Universal Robots PolyScope program: cinta.2.urp

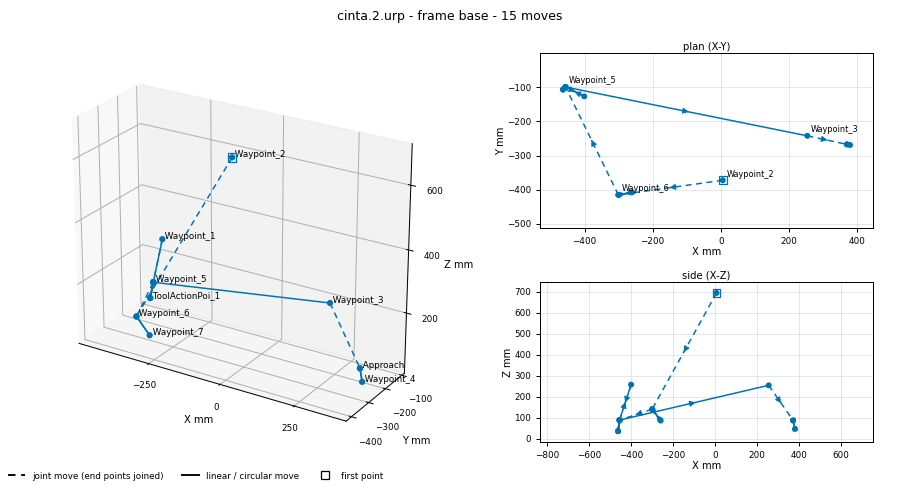
[picture p0: tool path of cinta.2.urp in frame base, 15 of 15 moves have a stored position in this frame; points joined in program order, loops and branches not executed]
Program cinta.2 (installation=default directory=/programs createdIn=5.14.5 lastSavedIn=5.14.5 robotSerialNumber=20195300809)
Calibrated DH parameters: a=[-0.000085, -0.20076, -0.212369, 0.000121, -0.000118, 0]; d=[0.15185, -26.306375, 24.753047, 1.684739, 0.085386, 0.092088]; alpha=[1.572149, -0.00522, -0.011864, 1.571339, -1.571085, 0]; deltaTheta=[0, 0.599885, -0.513355, -0.086555, 0.000006, 0]
InitVariablesNode variables(variable(name=Pallet_1_cnt_1, expression=1), variable(name=Pallet_1_lct, expression=1), variable(name=Pallet_1_lno, expression=1), variable(name=Pallet_1_sep, expression=False), variable(name=Pallet_1_tct, expression=1), variable(name=Pallet_2_cnt_1, expression=1), variable(name=Pallet_2_cnt_2, expression=1), variable(name=Pallet_2_lct, expression=1), variable(name=Pallet_2_lct_1, expression=1), variable(name=Pallet_2_lno, expression=1), variable(name=Pallet_2_lno_1, expression=1), variable(name=Pallet_2_sep, expression=False), variable(name=Pallet_2_sep_1, expression=False), variable(name=Pallet_2_tct, expression=1), variable(name=Pallet_2_tct_1, expression=1), variable(name=Pallet_4_cnt, expression=1), variable(name=Pallet_4_lct, expression=1), variable(name=Pallet_4_lno, expression=1), variable(name=Pallet_4_sep, expression=False), variable(name=Pallet_4_tct, expression=1))
Robot Program (runOnlyOnce=false)
  URCap Gripper Activate (Robotiq_Grippers, Robotiq Inc.) dataModel(ResetAndActivateKey=false)
  MoveJ speed 60 deg/s, acceleration 80 deg/s^2 (useActiveTCP=true) feature=Base
    Waypoint Waypoint_2: TCP in base x=5.936 y=-372.7 z=694.672 mm, rx=-0.0178 ry=2.2101 rz=-2.2165 rad; joints [0.003, -89.998, 0.001, -89.999, 0, 0.002] deg; TCP offset x=0 y=0 z=150 mm, rx=0 ry=0 rz=0 rad
  Wait DigitalInput pin=digital_in[0]; digitalValue=0
  URCap Palletizing (polyscope-pallet-impl, Universal Robots) dataModel(palletFeature=Base, isPalletizing=true, Variable(key=name, variable(name=Pallet_1)), Variable(key=globalCountingVariable, variable(name=Pallet_1_cnt_1, initializeExpression=1)), Variable(key=layerNumberVariable, variable(name=Pallet_1_lno, initializeExpression=1)), Variable(key=layerCountingVariable, variable(name=Pallet_1_lct, initializeExpression=1)), Variable(key=handleSeparatorVariable, variable(name=Pallet_1_sep, initializeExpression=False)), Variable(key=totalCountVariable, variable(name=Pallet_1_tct, initializeExpression=1)), Length(key=objectHeight value=0.04 unit=M), Variable(key=referencePoint, variable(featureName=referencePoint)), Variable(key=separatorPoint, variable(featureName=separatorPoint))); state(isChildrenLocked=true)
    URCap Patterns (polyscope-pallet-impl, Universal Robots) state(isChildrenLocked=true)
      URCap Pattern (polyscope-pallet-impl, Universal Robots) dataModel(UUID=7d18734c-cb0f-4b21-a534-5904a56affce, patternType=IRREGULAR, Variable(key=nameVariable, variable(name=Irreg_Pattern_1))); state(isChildrenLocked=true)
        URCap Item (polyscope-pallet-impl, Universal Robots) dataModel(UUID=f348ba63-6d21-43bb-8ae8-3964627112de, patternType=IRREGULAR, index=0, calibrationDeltaTheta=[2.0871938292282843E-8, 0.5998849625986696, -0.513354759222901, -0.08655474087847535, 6.239817607139875E-6, -6.658617090343766E-8], calibrationA=[-8.52060452638757E-5, -0.2007601879611388, -0.2123691625519033, 1.2105607098011576E-4, -1.1833705743435544E-4, 0.0], calibrationD=[0.15184970286177432, -26.306374840159272, 24.75304670983349, 1.6847390881089916, 0.085385969004481, 0.09208826337351553], calibrationAlpha=[1.5721487795181908, -0.005219907129425837, -0.011864150755780208, 1.5713392161993658, -1.5710853432049288, 0.0], calibrationJointChecksum=[-1860213401, -1859864814, -1494669377, -1328152407, -1329437658, -1329056899], calibrationStatus=2, calibrationValidChecksum=true, baseToFeature=[0.0, 0.0, 0.0, 0.0, 0.0, 0.0], TCPOffset=[9.391397651714595E-6, 1.2583319936476656E-5, 0.15002059384390531, -4.260528976040452E-5, 2.8840070067630035E-6, -1.0843116676403497E-6], Variable(key=variable, variable(name=Item_1)), JointPositions(key=jointpositions, JointPosition(key=[1], Angle(key=pos value=0.595677 unit=RAD)), JointPosition(key=[2], Angle(key=pos value=-0.675595 unit=RAD)), JointPosition(key=[3], Angle(key=pos value=0.603004 unit=RAD)), JointPosition(key=[4], Angle(key=pos value=-1.618024 unit=RAD)), JointPosition(key=[5], Angle(key=pos value=-1.472761 unit=RAD)), JointPosition(key=[6], Angle(key=pos value=-0.97685 unit=RAD))))
    URCap Layers (polyscope-pallet-impl, Universal Robots) dataModel(separators=[false], selectedPatterns=[7d18734c-cb0f-4b21-a534-5904a56affce])
    URCap At Each Item (polyscope-pallet-impl, Universal Robots) dataModel(selectedPattern=7d18734c-cb0f-4b21-a534-5904a56affce, selectedPosition=f348ba63-6d21-43bb-8ae8-3964627112de, Approach_calibrationDeltaTheta=[2.0871938292282843E-8, 0.5998849625986696, -0.513354759222901, -0.08655474087847535, 6.239817607139875E-6, -6.658617090343766E-8], Approach_calibrationA=[-8.52060452638757E-5, -0.2007601879611388, -0.2123691625519033, 1.2105607098011576E-4, -1.1833705743435544E-4, 0.0], Approach_calibrationD=[0.15184970286177432, -26.306374840159272, 24.75304670983349, 1.6847390881089916, 0.085385969004481, 0.09208826337351553], Approach_calibrationAlpha=[1.5721487795181908, -0.005219907129425837, -0.011864150755780208, 1.5713392161993658, -1.5710853432049288, 0.0], Approach_calibrationJointChecksum=[-1860213401, -1859864814, -1494669377, -1328152407, -1329437658, -1329056899], Approach_calibrationStatus=2, Approach_calibrationValidChecksum=true, Approach_baseToFeature=[0.0, 0.0, 0.0, 0.0, 0.0, 0.0], Approach_TCPOffset=[6.288453330560717E-6, -4.440500703251082E-6, 0.14999119071126726, 5.857466069426218E-5, -5.428145810996883E-6, 2.090200739322049E-5], Exit_calibrationDeltaTheta=[2.0871938292282843E-8, 0.5998849625986696, -0.513354759222901, -0.08655474087847535, 6.239817607139875E-6, -6.658617090343766E-8], Exit_calibrationA=[-8.52060452638757E-5, -0.2007601879611388, -0.2123691625519033, 1.2105607098011576E-4, -1.1833705743435544E-4, 0.0], Exit_calibrationD=[0.15184970286177432, -26.306374840159272, 24.75304670983349, 1.6847390881089916, 0.085385969004481, 0.09208826337351553], Exit_calibrationAlpha=[1.5721487795181908, -0.005219907129425837, -0.011864150755780208, 1.5713392161993658, -1.5710853432049288, 0.0], Exit_calibrationJointChecksum=[-1860213401, -1859864814, -1494669377, -1328152407, -1329437658, -1329056899], Exit_calibrationStatus=2, Exit_calibrationValidChecksum=true, Exit_baseToFeature=[0.0, 0.0, 0.0, 0.0, 0.0, 0.0], Exit_TCPOffset=[-1.7989367446957782E-5, -1.0560005302862052E-5, 0.15002098103245548, -3.476895864800672E-6, -4.621995147941492E-5, -3.533771160372287E-5], currentWizardState=LANDING, Pose(key=refBaseToFeature, Position(key=posePosition, Length(key=X value=0 unit=M), Length(key=Y value=0 unit=M), Length(key=Z value=0 unit=M)), Rotation(key=poseRotation, Angle(key=RX value=0 unit=RAD), Angle(key=RY value=0 unit=RAD), Angle(key=RZ value=0 unit=RAD))), Pose(key=refPose, Position(key=posePosition, Length(key=X value=-0.356569 unit=M), Length(key=Y value=-0.423777 unit=M), Length(key=Z value=0.09165 unit=M)), Rotation(key=poseRotation, Angle(key=RX value=0.142297 unit=RAD), Angle(key=RY value=-3.021243 unit=RAD), Angle(key=RZ value=0.176168 unit=RAD))), JointPositions(key=Approach_jointpositions, JointPosition(key=[1], Angle(key=pos value=0.546001 unit=RAD)), JointPosition(key=[2], Angle(key=pos value=-0.682183 unit=RAD)), JointPosition(key=[3], Angle(key=pos value=0.323504 unit=RAD)), JointPosition(key=[4], Angle(key=pos value=-1.411958 unit=RAD)), JointPosition(key=[5], Angle(key=pos value=-1.400218 unit=RAD)), JointPosition(key=[6], Angle(key=pos value=-1.026097 unit=RAD))), JointPositions(key=Exit_jointpositions, JointPosition(key=[1], Angle(key=pos value=0.615816 unit=RAD)), JointPosition(key=[2], Angle(key=pos value=-0.58775 unit=RAD)), JointPosition(key=[3], Angle(key=pos value=0.453411 unit=RAD)), JointPosition(key=[4], Angle(key=pos value=-1.593643 unit=RAD)), JointPosition(key=[5], Angle(key=pos value=-1.548909 unit=RAD)), JointPosition(key=[6], Angle(key=pos value=-1.048656 unit=RAD))))
      URCap Generated Movements (polyscope-pallet-impl, Universal Robots) state(isChildrenLocked=true)
        MoveJ speed 60 deg/s, acceleration 80 deg/s^2 (useActiveTCP=true) feature=referencePoint
          Waypoint Waypoint_6: TCP in base x=-300.88 y=-415.654 z=140.629 mm, rx=-0.0198 ry=-3.0249 rz=0.2808 rad; joints [36.906, -52.821, 49.281, -97.642, -86.084, -51.998] deg; feature pose in base x=-356.569 y=-423.777 z=91.65 mm, rx=0.1423 ry=-3.0212 rz=0.1762 rad
        MoveL speed 250 mm/s, acceleration 1200 mm/s^2 (useActiveTCP=true) feature(featureName=referencePoint)
          Waypoint Waypoint_7: TCP in base x=-260.278 y=-408.079 z=86.393 mm, rx=-0.0542 ry=-3.111 rz=0.0452 rad; joints [41.67, -49.638, 53.512, -96.276, -90.815, -46.427] deg
          SetPayload (workpieceName=Payload)
        Folder Tool action
          URCap Gripper (Robotiq_Grippers, Robotiq Inc.) dataModel(position=100.0, force=5.0, speed=100.0, positionInDouble=100.0, forceInDouble=5.0, speedInDouble=100.0, slaveIds=[3], blocking=true)
        MoveL speed 250 mm/s, acceleration 1200 mm/s^2 (useActiveTCP=true) feature(featureName=referencePoint)
          Waypoint Waypoint_6: TCP in base x=-300.88 y=-415.654 z=140.629 mm, rx=-0.0198 ry=-3.0249 rz=0.2808 rad; joints [36.906, -52.821, 49.281, -97.642, -86.084, -51.998] deg
  URCap Palletizing (polyscope-pallet-impl, Universal Robots) dataModel(palletFeature=Base, isPalletizing=false, Variable(key=name, variable(name=Pallet_2)), Variable(key=globalCountingVariable, variable(name=Pallet_2_cnt_1, initializeExpression=1)), Variable(key=layerNumberVariable, variable(name=Pallet_2_lno, initializeExpression=1)), Variable(key=layerCountingVariable, variable(name=Pallet_2_lct, initializeExpression=1)), Variable(key=handleSeparatorVariable, variable(name=Pallet_2_sep, initializeExpression=False)), Variable(key=totalCountVariable, variable(name=Pallet_2_tct, initializeExpression=1)), Length(key=objectHeight value=0.05 unit=M), Variable(key=referencePoint, variable(featureName=referencePoin_1)), Variable(key=separatorPoint, variable(featureName=separatorPoin_1))); state(isChildrenLocked=true)
    URCap Patterns (polyscope-pallet-impl, Universal Robots) state(isChildrenLocked=true)
      URCap Pattern (polyscope-pallet-impl, Universal Robots) dataModel(UUID=70c9da9f-f26c-40af-87f5-4ef85564398c, patternType=IRREGULAR, Variable(key=nameVariable, variable(name=Irreg_Pattern_2))); state(isChildrenLocked=true)
        URCap Item (polyscope-pallet-impl, Universal Robots) dataModel(UUID=c27a4a84-36a7-4a3e-9bbe-b9e4806bb6c1, patternType=IRREGULAR, index=0, calibrationDeltaTheta=[2.0871938292282843E-8, 0.5998849625986696, -0.513354759222901, -0.08655474087847535, 6.239817607139875E-6, -6.658617090343766E-8], calibrationA=[-8.52060452638757E-5, -0.2007601879611388, -0.2123691625519033, 1.2105607098011576E-4, -1.1833705743435544E-4, 0.0], calibrationD=[0.15184970286177432, -26.306374840159272, 24.75304670983349, 1.6847390881089916, 0.085385969004481, 0.09208826337351553], calibrationAlpha=[1.5721487795181908, -0.005219907129425837, -0.011864150755780208, 1.5713392161993658, -1.5710853432049288, 0.0], calibrationJointChecksum=[-1860213401, -1859864814, -1494669377, -1328152407, -1329437658, -1329056899], calibrationStatus=2, calibrationValidChecksum=true, baseToFeature=[0.0, 0.0, 0.0, 0.0, 0.0, 0.0], TCPOffset=[1.4796052247856295E-6, -1.2520157244955143E-5, 0.14999059913150856, 4.686731117752855E-5, -3.293405451311865E-5, 2.7796227253080194E-5], Variable(key=variable, variable(name=Item_2)), JointPositions(key=jointpositions, JointPosition(key=[1], Angle(key=pos value=-0.101307 unit=RAD)), JointPosition(key=[2], Angle(key=pos value=-0.846515 unit=RAD)), JointPosition(key=[3], Angle(key=pos value=1.123983 unit=RAD)), JointPosition(key=[4], Angle(key=pos value=-1.842057 unit=RAD)), JointPosition(key=[5], Angle(key=pos value=-1.498402 unit=RAD)), JointPosition(key=[6], Angle(key=pos value=-0.155893 unit=RAD))))
    URCap Layers (polyscope-pallet-impl, Universal Robots) dataModel(separators=[false], selectedPatterns=[70c9da9f-f26c-40af-87f5-4ef85564398c])
    URCap At Each Item (polyscope-pallet-impl, Universal Robots) dataModel(selectedPattern=70c9da9f-f26c-40af-87f5-4ef85564398c, selectedPosition=c27a4a84-36a7-4a3e-9bbe-b9e4806bb6c1, Approach_calibrationDeltaTheta=[2.0871938292282843E-8, 0.5998849625986696, -0.513354759222901, -0.08655474087847535, 6.239817607139875E-6, -6.658617090343766E-8], Approach_calibrationA=[-8.52060452638757E-5, -0.2007601879611388, -0.2123691625519033, 1.2105607098011576E-4, -1.1833705743435544E-4, 0.0], Approach_calibrationD=[0.15184970286177432, -26.306374840159272, 24.75304670983349, 1.6847390881089916, 0.085385969004481, 0.09208826337351553], Approach_calibrationAlpha=[1.5721487795181908, -0.005219907129425837, -0.011864150755780208, 1.5713392161993658, -1.5710853432049288, 0.0], Approach_calibrationJointChecksum=[-1860213401, -1859864814, -1494669377, -1328152407, -1329437658, -1329056899], Approach_calibrationStatus=2, Approach_calibrationValidChecksum=true, Approach_baseToFeature=[0.0, 0.0, 0.0, 0.0, 0.0, 0.0], Approach_TCPOffset=[-2.435285091917372E-6, -2.2477675725607327E-5, 0.14996372139900316, 1.2485897723616868E-4, 1.936593107412943E-5, -3.0361418856762723E-5], Exit_calibrationDeltaTheta=[2.0871938292282843E-8, 0.5998849625986696, -0.513354759222901, -0.08655474087847535, 6.239817607139875E-6, -6.658617090343766E-8], Exit_calibrationA=[-8.52060452638757E-5, -0.2007601879611388, -0.2123691625519033, 1.2105607098011576E-4, -1.1833705743435544E-4, 0.0], Exit_calibrationD=[0.15184970286177432, -26.306374840159272, 24.75304670983349, 1.6847390881089916, 0.085385969004481, 0.09208826337351553], Exit_calibrationAlpha=[1.5721487795181908, -0.005219907129425837, -0.011864150755780208, 1.5713392161993658, -1.5710853432049288, 0.0], Exit_calibrationJointChecksum=[-1860213401, -1859864814, -1494669377, -1328152407, -1329437658, -1329056899], Exit_calibrationStatus=2, Exit_calibrationValidChecksum=true, Exit_baseToFeature=[0.0, 0.0, 0.0, 0.0, 0.0, 0.0], Exit_TCPOffset=[1.7062831376105092E-5, 3.524481410888125E-6, 0.1500131622037378, -3.3427689265285523E-5, -7.770367597523134E-6, 3.124336029970859E-5], currentWizardState=LANDING, Pose(key=refBaseToFeature, Position(key=posePosition, Length(key=X value=0 unit=M), Length(key=Y value=0 unit=M), Length(key=Z value=0 unit=M)), Rotation(key=poseRotation, Angle(key=RX value=0 unit=RAD), Angle(key=RY value=0 unit=RAD), Angle(key=RZ value=0 unit=RAD))), Pose(key=refPose, Position(key=posePosition, Length(key=X value=-0.463666 unit=M), Length(key=Y value=-0.106221 unit=M), Length(key=Z value=0.035787 unit=M)), Rotation(key=poseRotation, Angle(key=RX value=2.122927 unit=RAD), Angle(key=RY value=2.233822 unit=RAD), Angle(key=RZ value=-0.100576 unit=RAD))), JointPositions(key=Approach_jointpositions, JointPosition(key=[1], Angle(key=pos value=-0.083249 unit=RAD)), JointPosition(key=[2], Angle(key=pos value=-0.988428 unit=RAD)), JointPosition(key=[3], Angle(key=pos value=1.052561 unit=RAD)), JointPosition(key=[4], Angle(key=pos value=-1.655373 unit=RAD)), JointPosition(key=[5], Angle(key=pos value=-1.48077 unit=RAD)), JointPosition(key=[6], Angle(key=pos value=-0.155884 unit=RAD))), JointPositions(key=Exit_jointpositions, JointPosition(key=[1], Angle(key=pos value=-0.101329 unit=RAD)), JointPosition(key=[2], Angle(key=pos value=-0.846523 unit=RAD)), JointPosition(key=[3], Angle(key=pos value=1.123971 unit=RAD)), JointPosition(key=[4], Angle(key=pos value=-1.842077 unit=RAD)), JointPosition(key=[5], Angle(key=pos value=-1.498362 unit=RAD)), JointPosition(key=[6], Angle(key=pos value=-0.155884 unit=RAD))))
      URCap Generated Movements (polyscope-pallet-impl, Universal Robots) state(isChildrenLocked=true)
        MoveJ speed 60 deg/s, acceleration 80 deg/s^2 (useActiveTCP=true) feature=referencePoin_1
          Waypoint Waypoint_5: TCP in base x=-456.282 y=-98.651 z=88.709 mm, rx=2.1005 ry=2.2182 rz=-0.0592 rad; joints [-6.749, -50.646, 52.859, -89.594, -86.16, -9.971] deg; feature pose in base x=-463.666 y=-106.221 z=35.787 mm, rx=2.1229 ry=2.2338 rz=-0.1006 rad
        MoveL speed 250 mm/s, acceleration 1200 mm/s^2 (useActiveTCP=true) feature(featureName=referencePoin_1)
          Waypoint ToolActionPoi_1: TCP in base x=-463.666 y=-106.221 z=35.787 mm, rx=2.1229 ry=2.2338 rz=-0.1006 rad; joints [-5.804, -48.502, 64.399, -105.542, -85.852, -8.932] deg; TCP offset x=0.001 y=-0.013 z=149.991 mm, rx=0 ry=0 rz=0 rad
        Folder Tool action
          URCap Gripper (Robotiq_Grippers, Robotiq Inc.) dataModel(position=0.0, force=100.0, speed=100.0, positionInDouble=0.0, forceInDouble=100.0, speedInDouble=100.0, slaveIds=[3], blocking=true)
        MoveL speed 250 mm/s, acceleration 1200 mm/s^2 (useActiveTCP=true) feature(featureName=referencePoin_1)
          Waypoint Waypoint_5: TCP in base x=-456.282 y=-98.651 z=88.709 mm, rx=2.1005 ry=2.2182 rz=-0.0592 rad; joints [-6.749, -50.646, 52.859, -89.594, -86.16, -9.971] deg; TCP offset x=0 y=0 z=150 mm, rx=0 ry=0 rz=0 rad
  MoveL speed 250 mm/s, acceleration 1200 mm/s^2 (useActiveTCP=true) feature=Base
    Waypoint Waypoint_1: TCP in base x=-401.164 y=-126.147 z=257.714 mm, rx=-2.0401 ry=-2.1933 rz=0.3328 rad; joints [-4.037, -76.934, 54.545, -81.338, -85.663, -7.38] deg
  Wait Sleep waitTime=3
  URCap Palletizing (polyscope-pallet-impl, Universal Robots) dataModel(palletFeature=Base, isPalletizing=false, Length(key=objectHeight value=0.05 unit=M), Variable(key=name, variable(name=Pallet_3)), Variable(key=globalCountingVariable, variable(name=Pallet_2_cnt_2, initializeExpression=1)), Variable(key=layerCountingVariable, variable(name=Pallet_2_lct_1, initializeExpression=1)), Variable(key=layerNumberVariable, variable(name=Pallet_2_lno_1, initializeExpression=1)), Variable(key=handleSeparatorVariable, variable(name=Pallet_2_sep_1, initializeExpression=False)), Variable(key=totalCountVariable, variable(name=Pallet_2_tct_1, initializeExpression=1)), Variable(key=referencePoint, variable(featureName=referencePoin_2)), Variable(key=separatorPoint, variable(featureName=separatorPoin_2))); state(isChildrenLocked=true)
    URCap Patterns (polyscope-pallet-impl, Universal Robots) state(isChildrenLocked=true)
      URCap Pattern (polyscope-pallet-impl, Universal Robots) dataModel(UUID=70c9da9f-f26c-40af-87f5-4ef85564398c, patternType=IRREGULAR, Variable(key=nameVariable, variable(name=Irreg_Pattern_3))); state(isChildrenLocked=true)
        URCap Item (polyscope-pallet-impl, Universal Robots) dataModel(UUID=c27a4a84-36a7-4a3e-9bbe-b9e4806bb6c1, patternType=IRREGULAR, index=0, calibrationDeltaTheta=[2.0871938292282843E-8, 0.5998849625986696, -0.513354759222901, -0.08655474087847535, 6.239817607139875E-6, -6.658617090343766E-8], calibrationA=[-8.52060452638757E-5, -0.2007601879611388, -0.2123691625519033, 1.2105607098011576E-4, -1.1833705743435544E-4, 0.0], calibrationD=[0.15184970286177432, -26.306374840159272, 24.75304670983349, 1.6847390881089916, 0.085385969004481, 0.09208826337351553], calibrationAlpha=[1.5721487795181908, -0.005219907129425837, -0.011864150755780208, 1.5713392161993658, -1.5710853432049288, 0.0], calibrationJointChecksum=[-1860213401, -1859864814, -1494669377, -1328152407, -1329437658, -1329056899], calibrationStatus=2, calibrationValidChecksum=true, baseToFeature=[0.0, 0.0, 0.0, 0.0, 0.0, 0.0], TCPOffset=[1.4796052247856295E-6, -1.2520157244955143E-5, 0.14999059913150856, 4.686731117752855E-5, -3.293405451311865E-5, 2.7796227253080194E-5], JointPositions(key=jointpositions, JointPosition(key=[1], Angle(key=pos value=-0.101307 unit=RAD)), JointPosition(key=[2], Angle(key=pos value=-0.846515 unit=RAD)), JointPosition(key=[3], Angle(key=pos value=1.123983 unit=RAD)), JointPosition(key=[4], Angle(key=pos value=-1.842057 unit=RAD)), JointPosition(key=[5], Angle(key=pos value=-1.498402 unit=RAD)), JointPosition(key=[6], Angle(key=pos value=-0.155893 unit=RAD))), Variable(key=variable, variable(name=Item_3)))
    URCap Layers (polyscope-pallet-impl, Universal Robots) dataModel(separators=[false], selectedPatterns=[70c9da9f-f26c-40af-87f5-4ef85564398c])
    URCap At Each Item (polyscope-pallet-impl, Universal Robots) dataModel(selectedPattern=70c9da9f-f26c-40af-87f5-4ef85564398c, selectedPosition=c27a4a84-36a7-4a3e-9bbe-b9e4806bb6c1, Approach_calibrationDeltaTheta=[2.0871938292282843E-8, 0.5998849625986696, -0.513354759222901, -0.08655474087847535, 6.239817607139875E-6, -6.658617090343766E-8], Approach_calibrationA=[-8.52060452638757E-5, -0.2007601879611388, -0.2123691625519033, 1.2105607098011576E-4, -1.1833705743435544E-4, 0.0], Approach_calibrationD=[0.15184970286177432, -26.306374840159272, 24.75304670983349, 1.6847390881089916, 0.085385969004481, 0.09208826337351553], Approach_calibrationAlpha=[1.5721487795181908, -0.005219907129425837, -0.011864150755780208, 1.5713392161993658, -1.5710853432049288, 0.0], Approach_calibrationJointChecksum=[-1860213401, -1859864814, -1494669377, -1328152407, -1329437658, -1329056899], Approach_calibrationStatus=2, Approach_calibrationValidChecksum=true, Approach_baseToFeature=[0.0, 0.0, 0.0, 0.0, 0.0, 0.0], Approach_TCPOffset=[-2.435285091917372E-6, -2.2477675725607327E-5, 0.14996372139900316, 1.2485897723616868E-4, 1.936593107412943E-5, -3.0361418856762723E-5], Exit_calibrationDeltaTheta=[2.0871938292282843E-8, 0.5998849625986696, -0.513354759222901, -0.08655474087847535, 6.239817607139875E-6, -6.658617090343766E-8], Exit_calibrationA=[-8.52060452638757E-5, -0.2007601879611388, -0.2123691625519033, 1.2105607098011576E-4, -1.1833705743435544E-4, 0.0], Exit_calibrationD=[0.15184970286177432, -26.306374840159272, 24.75304670983349, 1.6847390881089916, 0.085385969004481, 0.09208826337351553], Exit_calibrationAlpha=[1.5721487795181908, -0.005219907129425837, -0.011864150755780208, 1.5713392161993658, -1.5710853432049288, 0.0], Exit_calibrationJointChecksum=[-1860213401, -1859864814, -1494669377, -1328152407, -1329437658, -1329056899], Exit_calibrationStatus=2, Exit_calibrationValidChecksum=true, Exit_baseToFeature=[0.0, 0.0, 0.0, 0.0, 0.0, 0.0], Exit_TCPOffset=[1.7062831376105092E-5, 3.524481410888125E-6, 0.1500131622037378, -3.3427689265285523E-5, -7.770367597523134E-6, 3.124336029970859E-5], currentWizardState=LANDING, Pose(key=refBaseToFeature, Position(key=posePosition, Length(key=X value=0 unit=M), Length(key=Y value=0 unit=M), Length(key=Z value=0 unit=M)), Rotation(key=poseRotation, Angle(key=RX value=0 unit=RAD), Angle(key=RY value=0 unit=RAD), Angle(key=RZ value=0 unit=RAD))), Pose(key=refPose, Position(key=posePosition, Length(key=X value=-0.463666 unit=M), Length(key=Y value=-0.106221 unit=M), Length(key=Z value=0.035787 unit=M)), Rotation(key=poseRotation, Angle(key=RX value=2.122927 unit=RAD), Angle(key=RY value=2.233822 unit=RAD), Angle(key=RZ value=-0.100576 unit=RAD))), JointPositions(key=Approach_jointpositions, JointPosition(key=[1], Angle(key=pos value=-0.083249 unit=RAD)), JointPosition(key=[2], Angle(key=pos value=-0.988428 unit=RAD)), JointPosition(key=[3], Angle(key=pos value=1.052561 unit=RAD)), JointPosition(key=[4], Angle(key=pos value=-1.655373 unit=RAD)), JointPosition(key=[5], Angle(key=pos value=-1.48077 unit=RAD)), JointPosition(key=[6], Angle(key=pos value=-0.155884 unit=RAD))), JointPositions(key=Exit_jointpositions, JointPosition(key=[1], Angle(key=pos value=-0.101329 unit=RAD)), JointPosition(key=[2], Angle(key=pos value=-0.846523 unit=RAD)), JointPosition(key=[3], Angle(key=pos value=1.123971 unit=RAD)), JointPosition(key=[4], Angle(key=pos value=-1.842077 unit=RAD)), JointPosition(key=[5], Angle(key=pos value=-1.498362 unit=RAD)), JointPosition(key=[6], Angle(key=pos value=-0.155884 unit=RAD))))
      URCap Generated Movements (polyscope-pallet-impl, Universal Robots) state(isChildrenLocked=true)
        MoveJ speed 60 deg/s, acceleration 80 deg/s^2 (useActiveTCP=true) feature=referencePoin_2
          Waypoint Waypoint_5: TCP in base x=-456.282 y=-98.651 z=88.709 mm, rx=2.1005 ry=2.2182 rz=-0.0592 rad; joints [-6.749, -50.646, 52.859, -89.594, -86.16, -9.971] deg; feature pose in base x=-463.666 y=-106.221 z=35.787 mm, rx=2.1229 ry=2.2338 rz=-0.1006 rad
        MoveL speed 250 mm/s, acceleration 1200 mm/s^2 (useActiveTCP=true) feature(featureName=referencePoin_2)
          Waypoint ToolActionPoi_1: TCP in base x=-463.666 y=-106.221 z=35.787 mm, rx=2.1229 ry=2.2338 rz=-0.1006 rad; joints [-5.804, -48.502, 64.399, -105.542, -85.852, -8.932] deg; TCP offset x=0.001 y=-0.013 z=149.991 mm, rx=0 ry=0 rz=0 rad
        Folder Tool action
          URCap Gripper (Robotiq_Grippers, Robotiq Inc.) dataModel(position=100.0, force=5.0, speed=100.0, positionInDouble=100.0, forceInDouble=5.0, speedInDouble=100.0, slaveIds=[3], blocking=true)
        MoveL speed 250 mm/s, acceleration 1200 mm/s^2 (useActiveTCP=true) feature(featureName=referencePoin_2)
          Waypoint Waypoint_5: TCP in base x=-456.282 y=-98.651 z=88.709 mm, rx=2.1005 ry=2.2182 rz=-0.0592 rad; joints [-6.749, -50.646, 52.859, -89.594, -86.16, -9.971] deg; TCP offset x=0 y=0 z=150 mm, rx=0 ry=0 rz=0 rad
  MoveL speed 250 mm/s, acceleration 1200 mm/s^2 (useActiveTCP=true) feature=Base
    Waypoint Waypoint_3: TCP in base x=254.459 y=-242.142 z=254.509 mm, rx=0.8314 ry=-2.8675 rz=0.0376 rad; joints [120.819, -72.018, 40.908, -57.961, -99.758, -0.985] deg
  URCap Palletizing (polyscope-pallet-impl, Universal Robots) dataModel(palletFeature=Base, isPalletizing=true, Variable(key=name, variable(name=Pallet_4)), Variable(key=globalCountingVariable, variable(name=Pallet_4_cnt, initializeExpression=1)), Variable(key=layerNumberVariable, variable(name=Pallet_4_lno, initializeExpression=1)), Variable(key=layerCountingVariable, variable(name=Pallet_4_lct, initializeExpression=1)), Variable(key=handleSeparatorVariable, variable(name=Pallet_4_sep, initializeExpression=False)), Variable(key=totalCountVariable, variable(name=Pallet_4_tct, initializeExpression=1)), Length(key=objectHeight value=0.05 unit=M), Variable(key=referencePoint, variable(featureName=referencePoin_3)), Variable(key=separatorPoint, variable(featureName=separatorPoin_3))); state(isChildrenLocked=true)
    URCap Patterns (polyscope-pallet-impl, Universal Robots) state(isChildrenLocked=true)
      URCap Pattern (polyscope-pallet-impl, Universal Robots) dataModel(UUID=acebaf78-3d78-4eb2-9b5d-84c80f213af3, patternType=GRID, columns=3, rows=2, Variable(key=nameVariable, variable(name=Grid_Pattern_1))); state(isChildrenLocked=true)
        URCap Item (polyscope-pallet-impl, Universal Robots) dataModel(UUID=c01159d7-bdc8-4ad0-a768-e1fc64c23f72, patternType=GRID, index=0, calibrationDeltaTheta=[2.0871938292282843E-8, 0.5998849625986696, -0.513354759222901, -0.08655474087847535, 6.239817607139875E-6, -6.658617090343766E-8], calibrationA=[-8.52060452638757E-5, -0.2007601879611388, -0.2123691625519033, 1.2105607098011576E-4, -1.1833705743435544E-4, 0.0], calibrationD=[0.15184970286177432, -26.306374840159272, 24.75304670983349, 1.6847390881089916, 0.085385969004481, 0.09208826337351553], calibrationAlpha=[1.5721487795181908, -0.005219907129425837, -0.011864150755780208, 1.5713392161993658, -1.5710853432049288, 0.0], calibrationJointChecksum=[-1860213401, -1859864814, -1494669377, -1328152407, -1329437658, -1329056899], calibrationStatus=2, calibrationValidChecksum=true, baseToFeature=[0.0, 0.0, 0.0, 0.0, 0.0, 0.0], TCPOffset=[3.62221013627817E-7, 2.3695177266913614E-5, 0.14997395472124347, -8.099408147510325E-5, 4.151938501836787E-5, 1.2179441318642959E-5], Variable(key=variable, variable(name=CornerItem_1)), JointPositions(key=jointpositions, JointPosition(key=[1], Angle(key=pos value=2.248677 unit=RAD)), JointPosition(key=[2], Angle(key=pos value=-0.912649 unit=RAD)), JointPosition(key=[3], Angle(key=pos value=1.254868 unit=RAD)), JointPosition(key=[4], Angle(key=pos value=-1.946088 unit=RAD)), JointPosition(key=[5], Angle(key=pos value=-1.5722 unit=RAD)), JointPosition(key=[6], Angle(key=pos value=-2.450668 unit=RAD))))
        URCap Item (polyscope-pallet-impl, Universal Robots) dataModel(UUID=2189a120-c5c3-4d1a-9dea-873932fe821a, patternType=GRID, index=1, calibrationDeltaTheta=[2.0871938292282843E-8, 0.5998849625986696, -0.513354759222901, -0.08655474087847535, 6.239817607139875E-6, -6.658617090343766E-8], calibrationA=[-8.52060452638757E-5, -0.2007601879611388, -0.2123691625519033, 1.2105607098011576E-4, -1.1833705743435544E-4, 0.0], calibrationD=[0.15184970286177432, -26.306374840159272, 24.75304670983349, 1.6847390881089916, 0.085385969004481, 0.09208826337351553], calibrationAlpha=[1.5721487795181908, -0.005219907129425837, -0.011864150755780208, 1.5713392161993658, -1.5710853432049288, 0.0], calibrationJointChecksum=[-1860213401, -1859864814, -1494669377, -1328152407, -1329437658, -1329056899], calibrationStatus=2, calibrationValidChecksum=true, baseToFeature=[0.0, 0.0, 0.0, 0.0, 0.0, 0.0], TCPOffset=[6.919455813991782E-6, -1.59324717010495E-5, 0.15001367778842753, 2.9868797252186343E-5, -4.517849279249192E-6, -4.000161446948098E-5], Variable(key=variable, variable(name=CornerItem_2)), JointPositions(key=jointpositions, JointPosition(key=[1], Angle(key=pos value=2.614511 unit=RAD)), JointPosition(key=[2], Angle(key=pos value=-1.15318 unit=RAD)), JointPosition(key=[3], Angle(key=pos value=1.678785 unit=RAD)), JointPosition(key=[4], Angle(key=pos value=-2.080078 unit=RAD)), JointPosition(key=[5], Angle(key=pos value=-1.587274 unit=RAD)), JointPosition(key=[6], Angle(key=pos value=-2.091675 unit=RAD))))
        URCap Item (polyscope-pallet-impl, Universal Robots) dataModel(UUID=21607d58-3b12-46c5-8d2a-9916ff338648, patternType=GRID, index=2, calibrationDeltaTheta=[2.0871938292282843E-8, 0.5998849625986696, -0.513354759222901, -0.08655474087847535, 6.239817607139875E-6, -6.658617090343766E-8], calibrationA=[-8.52060452638757E-5, -0.2007601879611388, -0.2123691625519033, 1.2105607098011576E-4, -1.1833705743435544E-4, 0.0], calibrationD=[0.15184970286177432, -26.306374840159272, 24.75304670983349, 1.6847390881089916, 0.085385969004481, 0.09208826337351553], calibrationAlpha=[1.5721487795181908, -0.005219907129425837, -0.011864150755780208, 1.5713392161993658, -1.5710853432049288, 0.0], calibrationJointChecksum=[-1860213401, -1859864814, -1494669377, -1328152407, -1329437658, -1329056899], calibrationStatus=2, calibrationValidChecksum=true, baseToFeature=[0.0, 0.0, 0.0, 0.0, 0.0, 0.0], TCPOffset=[-4.63084492346999E-6, -4.863462618229231E-6, 0.1499865178152125, -7.754704754451109E-6, 1.2068952613309615E-6, 1.5530771283901447E-5], Variable(key=variable, variable(name=CornerItem_3)), JointPositions(key=jointpositions, JointPosition(key=[1], Angle(key=pos value=2.74226 unit=RAD)), JointPosition(key=[2], Angle(key=pos value=-0.741952 unit=RAD)), JointPosition(key=[3], Angle(key=pos value=0.93023 unit=RAD)), JointPosition(key=[4], Angle(key=pos value=-1.780847 unit=RAD)), JointPosition(key=[5], Angle(key=pos value=-1.58849 unit=RAD)), JointPosition(key=[6], Angle(key=pos value=-1.919331 unit=RAD))))
        URCap Item (polyscope-pallet-impl, Universal Robots) dataModel(UUID=203bc53d-136e-47a2-98ac-824ae0b9f02c, patternType=GRID, index=3, calibrationDeltaTheta=[2.0871938292282843E-8, 0.5998849625986696, -0.513354759222901, -0.08655474087847535, 6.239817607139875E-6, -6.658617090343766E-8], calibrationA=[-8.52060452638757E-5, -0.2007601879611388, -0.2123691625519033, 1.2105607098011576E-4, -1.1833705743435544E-4, 0.0], calibrationD=[0.15184970286177432, -26.306374840159272, 24.75304670983349, 1.6847390881089916, 0.085385969004481, 0.09208826337351553], calibrationAlpha=[1.5721487795181908, -0.005219907129425837, -0.011864150755780208, 1.5713392161993658, -1.5710853432049288, 0.0], calibrationJointChecksum=[-1860213401, -1859864814, -1494669377, -1328152407, -1329437658, -1329056899], calibrationStatus=2, calibrationValidChecksum=true, baseToFeature=[0.0, 0.0, 0.0, 0.0, 0.0, 0.0], TCPOffset=[2.9663871770058137E-6, -2.7200211151962028E-5, 0.15001295968752965, 2.8669519702431683E-5, -3.4484229554148914E-5, -1.2084844145554098E-5], Variable(key=variable, variable(name=CornerItem_4)), JointPositions(key=jointpositions, JointPosition(key=[1], Angle(key=pos value=2.423566 unit=RAD)), JointPosition(key=[2], Angle(key=pos value=-0.509839 unit=RAD)), JointPosition(key=[3], Angle(key=pos value=0.540103 unit=RAD)), JointPosition(key=[4], Angle(key=pos value=-1.69904 unit=RAD)), JointPosition(key=[5], Angle(key=pos value=-1.581203 unit=RAD)), JointPosition(key=[6], Angle(key=pos value=-2.232232 unit=RAD))))
    URCap Layers (polyscope-pallet-impl, Universal Robots) dataModel(separators=[false], selectedPatterns=[acebaf78-3d78-4eb2-9b5d-84c80f213af3])
    URCap At Each Item (polyscope-pallet-impl, Universal Robots) dataModel(selectedPattern=acebaf78-3d78-4eb2-9b5d-84c80f213af3, selectedPosition=c01159d7-bdc8-4ad0-a768-e1fc64c23f72, Approach_calibrationDeltaTheta=[2.0871938292282843E-8, 0.5998849625986696, -0.513354759222901, -0.08655474087847535, 6.239817607139875E-6, -6.658617090343766E-8], Approach_calibrationA=[-8.52060452638757E-5, -0.2007601879611388, -0.2123691625519033, 1.2105607098011576E-4, -1.1833705743435544E-4, 0.0], Approach_calibrationD=[0.15184970286177432, -26.306374840159272, 24.75304670983349, 1.6847390881089916, 0.085385969004481, 0.09208826337351553], Approach_calibrationAlpha=[1.5721487795181908, -0.005219907129425837, -0.011864150755780208, 1.5713392161993658, -1.5710853432049288, 0.0], Approach_calibrationJointChecksum=[-1860213401, -1859864814, -1494669377, -1328152407, -1329437658, -1329056899], Approach_calibrationStatus=2, Approach_calibrationValidChecksum=true, Approach_baseToFeature=[0.0, 0.0, 0.0, 0.0, 0.0, 0.0], Approach_TCPOffset=[-1.4970444630779678E-5, -1.8355945709314092E-5, 0.15001166807398744, 2.0599044056208026E-5, -2.093205654096037E-5, -3.220405087150925E-5], Exit_calibrationDeltaTheta=[2.0871938292282843E-8, 0.5998849625986696, -0.513354759222901, -0.08655474087847535, 6.239817607139875E-6, -6.658617090343766E-8], Exit_calibrationA=[-8.52060452638757E-5, -0.2007601879611388, -0.2123691625519033, 1.2105607098011576E-4, -1.1833705743435544E-4, 0.0], Exit_calibrationD=[0.15184970286177432, -26.306374840159272, 24.75304670983349, 1.6847390881089916, 0.085385969004481, 0.09208826337351553], Exit_calibrationAlpha=[1.5721487795181908, -0.005219907129425837, -0.011864150755780208, 1.5713392161993658, -1.5710853432049288, 0.0], Exit_calibrationJointChecksum=[-1860213401, -1859864814, -1494669377, -1328152407, -1329437658, -1329056899], Exit_calibrationStatus=2, Exit_calibrationValidChecksum=true, Exit_baseToFeature=[0.0, 0.0, 0.0, 0.0, 0.0, 0.0], Exit_TCPOffset=[3.322691039087111E-6, 1.1128758255485316E-5, 0.15000646305274576, -4.464457194953362E-5, 7.328457483196232E-6, -2.9105190136105157E-5], currentWizardState=SHOW_DONE, Pose(key=refBaseToFeature, Position(key=posePosition, Length(key=X value=0 unit=M), Length(key=Y value=0 unit=M), Length(key=Z value=0 unit=M)), Rotation(key=poseRotation, Angle(key=RX value=0 unit=RAD), Angle(key=RY value=0 unit=RAD), Angle(key=RZ value=0 unit=RAD))), Pose(key=refPose, Position(key=posePosition, Length(key=X value=0.368903 unit=M), Length(key=Y value=-0.26597 unit=M), Length(key=Z value=0.03651 unit=M)), Rotation(key=poseRotation, Angle(key=RX value=2.247353 unit=RAD), Angle(key=RY value=-2.156111 unit=RAD), Angle(key=RZ value=-0.085275 unit=RAD))), JointPositions(key=Approach_jointpositions, JointPosition(key=[1], Angle(key=pos value=2.227555 unit=RAD)), JointPosition(key=[2], Angle(key=pos value=-0.926507 unit=RAD)), JointPosition(key=[3], Angle(key=pos value=1.006304 unit=RAD)), JointPosition(key=[4], Angle(key=pos value=-1.626099 unit=RAD)), JointPosition(key=[5], Angle(key=pos value=-1.591359 unit=RAD)), JointPosition(key=[6], Angle(key=pos value=-0.911324 unit=RAD))), JointPositions(key=Exit_jointpositions, JointPosition(key=[1], Angle(key=pos value=2.241829 unit=RAD)), JointPosition(key=[2], Angle(key=pos value=-0.861087 unit=RAD)), JointPosition(key=[3], Angle(key=pos value=1.125595 unit=RAD)), JointPosition(key=[4], Angle(key=pos value=-1.784934 unit=RAD)), JointPosition(key=[5], Angle(key=pos value=-1.618915 unit=RAD)), JointPosition(key=[6], Angle(key=pos value=-0.942893 unit=RAD))))
      URCap Generated Movements (polyscope-pallet-impl, Universal Robots) state(isChildrenLocked=true)
        MoveJ speed 60 deg/s, acceleration 80 deg/s^2 (useActiveTCP=true) feature=referencePoin_3
          Waypoint Approach: TCP in base x=370.762 y=-267.292 z=87.108 mm, rx=2.2164 ry=-2.2232 rz=-0.0396 rad; joints [127.63, -53.085, 57.657, -93.169, -91.178, -52.215] deg; TCP offset x=-0.015 y=-0.018 z=150.012 mm, rx=0 ry=0 rz=0 rad; feature pose in base x=368.903 y=-265.97 z=36.51 mm, rx=2.2474 ry=-2.1561 rz=-0.0853 rad
        MoveL speed 250 mm/s, acceleration 1200 mm/s^2 (useActiveTCP=true) feature(featureName=referencePoin_3)
          Waypoint Waypoint_4: TCP in base x=379.925 y=-269.103 z=46.926 mm, rx=2.2216 ry=-2.1408 rz=-0.1246 rad; joints [130.192, -44.839, 53.206, -94.096, -94.423, -51.868] deg; TCP offset x=0 y=0 z=150 mm, rx=0 ry=0 rz=0 rad
        Folder Tool action
          URCap Gripper (Robotiq_Grippers, Robotiq Inc.) dataModel(position=0.0, force=100.0, speed=100.0, positionInDouble=0.0, forceInDouble=100.0, speedInDouble=100.0, slaveIds=[3], blocking=true)
        MoveL speed 250 mm/s, acceleration 1200 mm/s^2 (useActiveTCP=true) feature(featureName=referencePoin_3)
          Waypoint Approach: TCP in base x=370.762 y=-267.292 z=87.108 mm, rx=2.2164 ry=-2.2232 rz=-0.0396 rad; joints [127.63, -53.085, 57.657, -93.169, -91.178, -52.215] deg; TCP offset x=-0.015 y=-0.018 z=150.012 mm, rx=0 ry=0 rz=0 rad
Thread Thread_1 (runOnlyOnce=false)
  If digital_in[0]≠0 (checkContinuously=true)
    Set DigitalOutput pin=digital_out[0]; digitalValue=1
  Else 
    Set DigitalOutput pin=digital_out[0]; digitalValue=0
